% RSLogix 500 project P2_IVANOVSKI_M.RSS, saved by version 8.30.00.16 %
PROJECT "UNTITLED"    % processor: Bul.1763 MicroLogix 1100 Series B %

PROGRAM FILES
  LAD 2 "MAIN"  3 rungs
  LAD 3 "DIGITAL IO"  8 rungs
  LAD 4 "CONTROLS"  11 rungs

DATA FILES
  O0 OUTPUT  5 elements
  I1 INPUT  7 elements
  S2 STATUS  66 elements
  B3 BINARY  2 elements
  T4 TIMER  2 elements
  C5 COUNTER  1 elements
  R6 CONTROL  1 elements
  N7 INTEGER  6 elements
  F8 FLOAT  1 elements

LADDER 2 "MAIN"
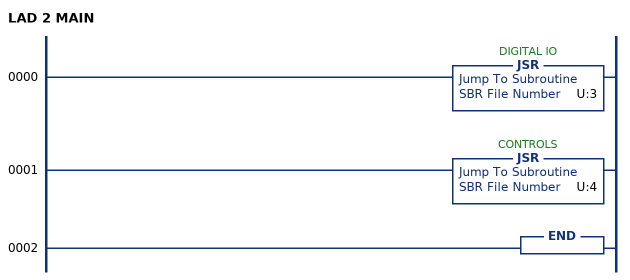
% Rung: 0 %
SOR JSR U:3 EOR
%   U:3  "DIGITAL IO" %
% Rung: 1 %
SOR JSR U:4 EOR
%   U:4  "CONTROLS" %
% Rung: 2 %
SOR END EOR

LADDER 3 "DIGITAL IO"
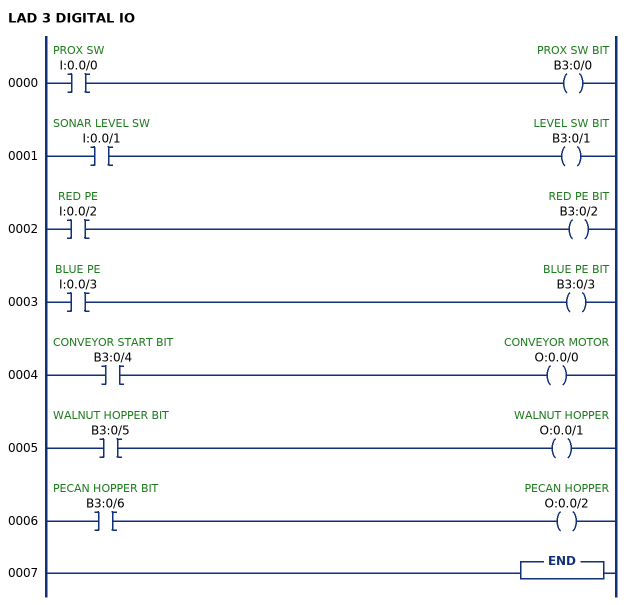
% Rung: 0 %
SOR XIC I:0.0/0 OTE B3:0/0 EOR
%   I:0.0/0  "PROX SW" %
%   B3:0/0  "PROX SW BIT" %
% Rung: 1 %
SOR XIC I:0.0/1 OTE B3:0/1 EOR
%   I:0.0/1  "SONAR LEVEL SW" %
%   B3:0/1  "LEVEL SW BIT" %
% Rung: 2 %
SOR XIC I:0.0/2 OTE B3:0/2 EOR
%   I:0.0/2  "RED PE" %
%   B3:0/2  "RED PE BIT" %
% Rung: 3 %
SOR XIC I:0.0/3 OTE B3:0/3 EOR
%   I:0.0/3  "BLUE PE" %
%   B3:0/3  "BLUE PE BIT" %
% Rung: 4 %
SOR XIC B3:0/4 OTE O:0.0/0 EOR
%   B3:0/4  "CONVEYOR START BIT" %
%   O:0.0/0  "CONVEYOR MOTOR" %
% Rung: 5 %
SOR XIC B3:0/5 OTE O:0.0/1 EOR
%   B3:0/5  "WALNUT HOPPER BIT" %
%   O:0.0/1  "WALNUT HOPPER" %
% Rung: 6 %
SOR XIC B3:0/6 OTE O:0.0/2 EOR
%   B3:0/6  "PECAN HOPPER BIT" %
%   O:0.0/2  "PECAN HOPPER" %
% Rung: 7 %
SOR END EOR

LADDER 4 "CONTROLS"
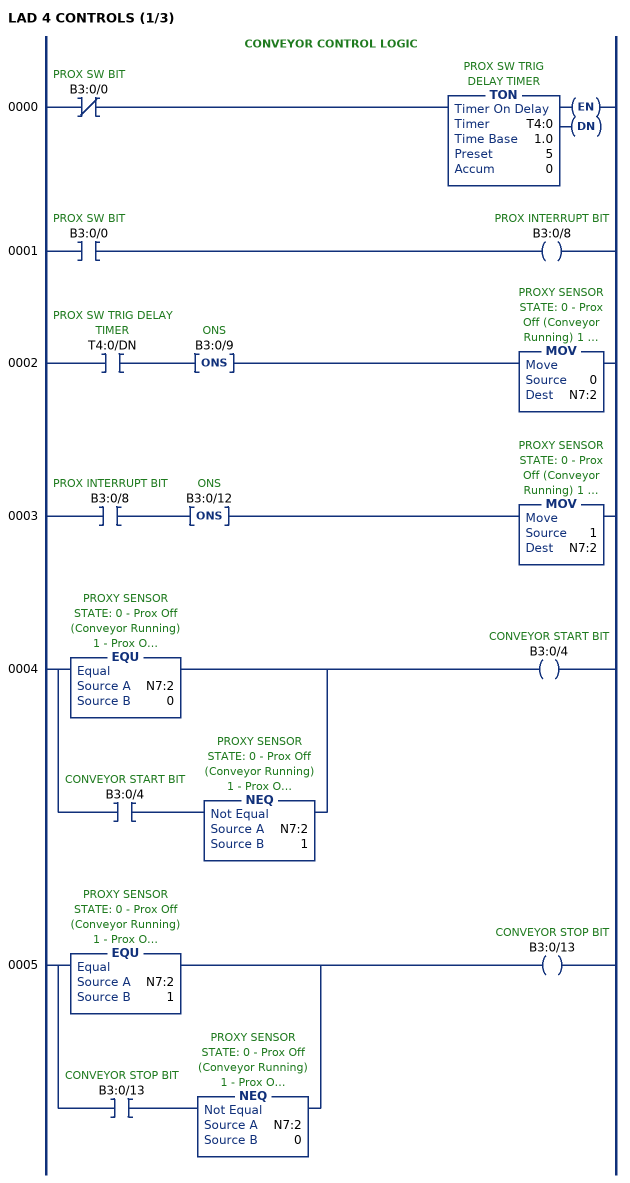
% Rung: 0 %
% TITLE: CONVEYOR CONTROL LOGIC %
SOR XIO B3:0/0 TON T4:0 1.0 5 0 EOR
%   B3:0/0  "PROX SW BIT" %
%   T4:0  "PROX SW TRIG DELAY TIMER" %
% Rung: 1 %
SOR XIC B3:0/0 OTE B3:0/8 EOR
%   B3:0/0  "PROX SW BIT" %
%   B3:0/8  "PROX INTERRUPT BIT" %
% Rung: 2 %
SOR XIC T4:0/DN ONS B3:0/9 MOV 0 N7:2 EOR
%   T4:0  "PROX SW TRIG DELAY TIMER" %
%   B3:0/9  "ONS" %
%   N7:2  "PROXY SENSOR STATE: 0 - Prox Off (Conveyor Running) 1 - Prox On (Conveyor Stopped)" %
% Rung: 3 %
SOR XIC B3:0/8 ONS B3:0/12 MOV 1 N7:2 EOR
%   B3:0/8  "PROX INTERRUPT BIT" %
%   B3:0/12  "ONS" %
%   N7:2  "PROXY SENSOR STATE: 0 - Prox Off (Conveyor Running) 1 - Prox On (Conveyor Stopped)" %
% Rung: 4 %
SOR BST EQU N7:2 0 NXB XIC B3:0/4 NEQ N7:2 1 BND OTE B3:0/4 EOR
%   N7:2  "PROXY SENSOR STATE: 0 - Prox Off (Conveyor Running) 1 - Prox On (Conveyor Stopped)" %
%   B3:0/4  "CONVEYOR START BIT" %
% Rung: 5 %
SOR BST EQU N7:2 1 NXB XIC B3:0/13 NEQ N7:2 0 BND OTE B3:0/13 EOR
%   N7:2  "PROXY SENSOR STATE: 0 - Prox Off (Conveyor Running) 1 - Prox On (Conveyor Stopped)" %
%   B3:0/13  "CONVEYOR STOP BIT" %

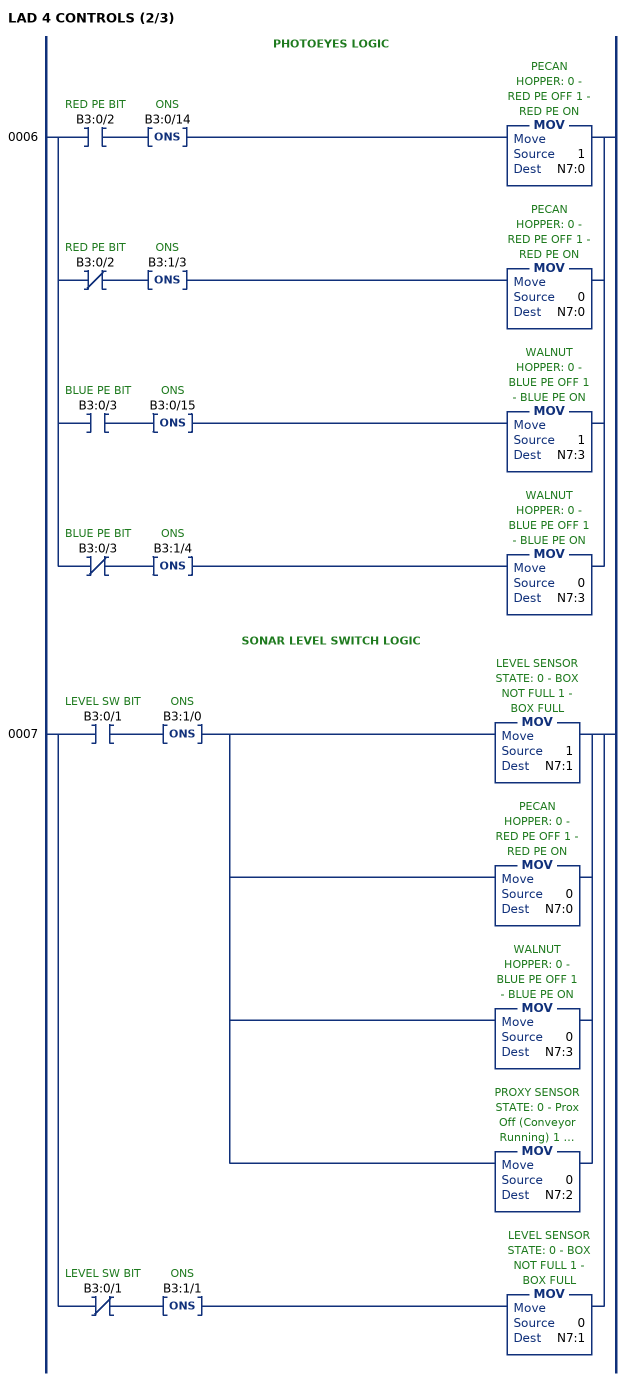
% Rung: 6 %
% TITLE: PHOTOEYES LOGIC %
SOR BST XIC B3:0/2 ONS B3:0/14 MOV 1 N7:0 NXB XIO B3:0/2 ONS B3:1/3 MOV 0 N7:0 NXB XIC B3:0/3 ONS B3:0/15 MOV 1 N7:3 NXB XIO B3:0/3 ONS B3:1/4 MOV 0 N7:3 BND EOR
%   B3:0/2  "RED PE BIT" %
%   B3:0/14  "ONS" %
%   N7:0  "PECAN HOPPER: 0 - RED PE OFF 1 - RED PE ON" %
%   B3:1/3  "ONS" %
%   B3:0/3  "BLUE PE BIT" %
%   B3:0/15  "ONS" %
%   N7:3  "WALNUT HOPPER: 0 - BLUE PE OFF 1 - BLUE PE ON" %
%   B3:1/4  "ONS" %
% Rung: 7 %
% TITLE: SONAR LEVEL SWITCH LOGIC %
SOR BST XIC B3:0/1 ONS B3:1/0 BST MOV 1 N7:1 NXB MOV 0 N7:0 NXB MOV 0 N7:3 NXB MOV 0 N7:2 BND NXB XIO B3:0/1 ONS B3:1/1 MOV 0 N7:1 BND EOR
%   B3:0/1  "LEVEL SW BIT" %
%   B3:1/0  "ONS" %
%   N7:1  "LEVEL SENSOR STATE: 0 - BOX NOT FULL 1 - BOX FULL" %
%   N7:0  "PECAN HOPPER: 0 - RED PE OFF 1 - RED PE ON" %
%   N7:3  "WALNUT HOPPER: 0 - BLUE PE OFF 1 - BLUE PE ON" %
%   N7:2  "PROXY SENSOR STATE: 0 - Prox Off (Conveyor Running) 1 - Prox On (Conveyor Stopped)" %
%   B3:1/1  "ONS" %

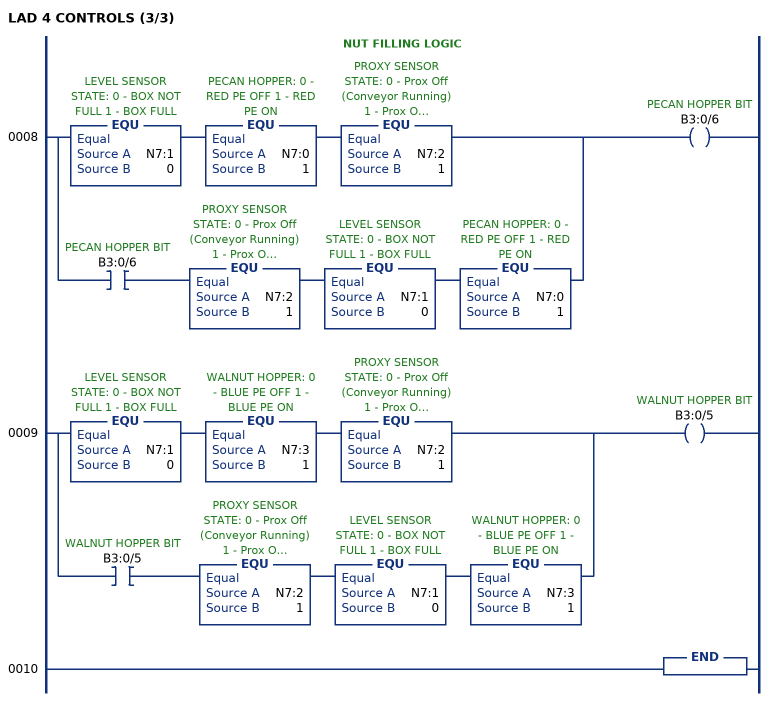
% Rung: 8 %
% TITLE: NUT FILLING LOGIC %
SOR BST EQU N7:1 0 EQU N7:0 1 EQU N7:2 1 NXB XIC B3:0/6 EQU N7:2 1 EQU N7:1 0 EQU N7:0 1 BND OTE B3:0/6 EOR
%   N7:1  "LEVEL SENSOR STATE: 0 - BOX NOT FULL 1 - BOX FULL" %
%   N7:0  "PECAN HOPPER: 0 - RED PE OFF 1 - RED PE ON" %
%   N7:2  "PROXY SENSOR STATE: 0 - Prox Off (Conveyor Running) 1 - Prox On (Conveyor Stopped)" %
%   B3:0/6  "PECAN HOPPER BIT" %
% Rung: 9 %
SOR BST EQU N7:1 0 EQU N7:3 1 EQU N7:2 1 NXB XIC B3:0/5 EQU N7:2 1 EQU N7:1 0 EQU N7:3 1 BND OTE B3:0/5 EOR
%   N7:1  "LEVEL SENSOR STATE: 0 - BOX NOT FULL 1 - BOX FULL" %
%   N7:3  "WALNUT HOPPER: 0 - BLUE PE OFF 1 - BLUE PE ON" %
%   N7:2  "PROXY SENSOR STATE: 0 - Prox Off (Conveyor Running) 1 - Prox On (Conveyor Stopped)" %
%   B3:0/5  "WALNUT HOPPER BIT" %
% Rung: 10 %
SOR END EOR

OTHER DOCUMENTED ADDRESSES
  B3:0/7  "PROX TRIGGER"
  B3:0/10  "CONVEYOR TRIGGER"
  B3:0/11  "PROX INTERRUPT"
  B3:1/2  "ONS"
  N7:4  "3 - Red PE OFF 4 - Blue PE OFF 5 - Both PEs OFF"
  N7:5  "3 - Red PE OFF 4 - Blue PE OFF 5 - Both PEs OFF"
  T4:1  "PROX SW INTERRUPT DELAY TIMER"

DATA TABLE (non-zero values as saved)
DATA T4
% .PRE .ACC %
% T4:0 % 5 0
% T4:1 % 3 0
